{attribute addProperty BoxType "EJ1957-0000-0017"}
{attribute addProperty Id "WcState0AT %I*BIT10.1250WcState1AT %I*BIT10.1250InputToggle0AT %I*BIT10.1250InputToggle1AT %I*BIT10.1250"}
{attribute addProperty CRC "3701249813"}
{attribute addProperty SizeInBites "4"}
{attribute addProperty SizeInBytes "0.5"}
TYPE WcState_DC9C9715 :
STRUCT
	{attribute addProperty Name "WcState0"}
	WcState0 AT %I* : BOOL;
	{attribute addProperty Name "WcState1"}
	WcState1 AT %I* : BOOL;
	{attribute addProperty Name "InputToggle0"}
	InputToggle0 AT %I* : BOOL;
	{attribute addProperty Name "InputToggle1"}
	InputToggle1 AT %I* : BOOL;
END_STRUCT
END_TYPE

(* stored: Version 1.2.0.0, ProductVersion 3.1.4024.9
   DUT WcState_DC9C9715: Id {14c2622f-6397-4458-a9e7-e08cbae00159} *)
